# EPICS substitutions: ek9000App/Db/EL1018.substitutions
file EL1018.template
{ 	pattern
	{
		TERMINAL,

	}
	{
	}
}
